Universal Robots PolyScope program: TFM_MAU.urp

Program TFM_MAU (installation=TFM_MAU directory=/programs/usbdisk createdIn=5.11.5.1010327 lastSavedIn=5.11.5.1010327 robotSerialNumber=20215301076)
Calibrated DH parameters: a=[-0.00009, -0.213549, -0.209038, 0.000077, -0.000166, 0]; d=[0.151848, 64.217848, -61.640034, -2.447154, 0.085569, 0.092371]; alpha=[1.570043, -0.001832, 0.017213, 1.572481, -1.574049, 0]; deltaTheta=[0, -0.503479, 0.712611, -0.209158, -0.000004, -0.000001]
Robot Program (runOnlyOnce=false)
  URCap Zimmer (Z_Gripper_C, Zimmer Group) dataModel(gripper_installation_scheme=257, gripper_number=3, program_number=1, program_name=Z_Release, program_settings=264)
  URCap External Control (External Control, FZI Research Center for Information Technology)
  URCap Zimmer (Z_Gripper_C, Zimmer Group) dataModel(gripper_installation_scheme=257, gripper_number=3, program_number=2, program_name=Z_Grip, program_settings=264)
  Wait Sleep waitTime=5
  URCap External Control (External Control, FZI Research Center for Information Technology)
  URCap Zimmer (Z_Gripper_C, Zimmer Group) dataModel(gripper_installation_scheme=257, gripper_number=3, program_number=1, program_name=Z_Release, program_settings=264)
  Wait Sleep waitTime=5
  URCap External Control (External Control, FZI Research Center for Information Technology)
